ABB RobotStudio station: Vision_HG_20240222-084128.rsstn

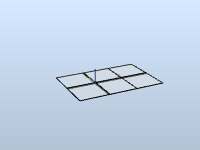
Station Station (saved by RobotStudio 6.8.8148.134)
Layout (positions relative to the parent item):
  - 框架_2 [frame] at (695.76, -308.93, 242.8) mm, rotated rx -4.43 ry -84.98 rz 46.15 deg
